(* IEC 61131-3 sources: repolevel_ST_code_completion/output/0127完整版本_带planner/repoeval_VisuElements/readful_result_no_provide, 3 files *)

(* ---- MouseEventHandler.st ---- *)
VAR
    LeftClickTimer : TON;
    xLeftClickOld : BOOL;
    iClickCount : INT := 0;
    xEventProcessed : BOOL := FALSE;
    rLastMouseX : REAL := 0.0;
    rLastMouseY : REAL := 0.0;
END_VAR

(* Reset event state *)
eMouseEvent := 0;
xEventActive := FALSE;

(* Handle left click events (single/double click) *)
IF xLeftClick AND NOT xLeftClickOld THEN
    (* First click detected *)
    IF iClickCount = 0 THEN
        LeftClickTimer(IN := TRUE, PT := tDblClickTime);
        iClickCount := 1;
    ELSE
        (* Second click within time window *)
        LeftClickTimer(IN := FALSE);
        eMouseEvent := 2; (* Double click *)
        rEventX := rMouseX;
        rEventY := rMouseY;
        xEventActive := TRUE;
        iClickCount := 0;
        xEventProcessed := TRUE;
    END_IF
ELSIF NOT xLeftClick AND xLeftClickOld THEN
    (* Left button released *)
    IF iClickCount = 1 AND NOT xEventProcessed THEN
        LeftClickTimer();
        IF NOT LeftClickTimer.Q THEN
            (* Still waiting for potential double click *)
        ELSE
            (* Timeout, register single click *)
            eMouseEvent := 1; (* Single click *)
            rEventX := rMouseX;
            rEventY := rMouseY;
            xEventActive := TRUE;
            iClickCount := 0;
        END_IF
    END_IF
END_IF

(* Check for double click timeout *)
IF LeftClickTimer.Q AND iClickCount = 1 THEN
    (* Timeout, register single click *)
    eMouseEvent := 1; (* Single click *)
    rEventX := rMouseX;
    rEventY := rMouseY;
    xEventActive := TRUE;
    iClickCount := 0;
END_IF

(* Handle right click events *)
IF xRightClick THEN
    eMouseEvent := 3; (* Right click *)
    rEventX := rMouseX;
    rEventY := rMouseY;
    xEventActive := TRUE;
END_IF

(* Handle middle click events *)
IF xMiddleClick THEN
    eMouseEvent := 4; (* Middle click *)
    rEventX := rMouseX;
    rEventY := rMouseY;
    xEventActive := TRUE;
END_IF

(* Handle mouse movement events *)
IF xMouseMove AND (rMouseX <> rLastMouseX OR rMouseY <> rLastMouseY) THEN
    eMouseEvent := 0; (* Mouse move *)
    rEventX := rMouseX;
    rEventY := rMouseY;
    xEventActive := TRUE;
    rLastMouseX := rMouseX;
    rLastMouseY := rMouseY;
END_IF

(* Update old state *)
xLeftClickOld := xLeftClick;
END_FUNCTION_BLOCK

(* ---- NodeExpandCollapse.st ---- *)
VAR
    NodeDblClick : TON; (* Timer for detecting double click *)
    xNodeClickOld : BOOL; (* Previous state of the click input *)
    iNodeState : INT := 1; (* State machine variable *)
END_VAR

CASE iNodeState OF

    1: (* Wait for first click *)
        IF xNodeClick AND NOT xNodeClickOld THEN
            NodeDblClick(IN := TRUE, PT := tDblClickTime);
            iNodeState := 2;
            xNodeSelected := TRUE;
        END_IF

    2: (* Wait for second click or timeout *)
        NodeDblClick();
        IF NodeDblClick.Q THEN
            (* Timeout - single click, reset *)
            NodeDblClick(IN := FALSE);
            xNodeClickOld := FALSE;
            iNodeState := 1;
            xNodeSelected := FALSE;
        ELSIF NOT xNodeClick AND xNodeClickOld THEN
            (* Second click detected - toggle expansion *)
            NodeDblClick(IN := FALSE);
            xNodeExpand := NOT xNodeExpand;
            iNodeState := 1;
            xNodeSelected := FALSE;
        END_IF

END_CASE

xNodeClickOld := xNodeClick;
END_FUNCTION_BLOCK

(* ---- RotationCalculation.st ---- *)
VAR
    rRadians : REAL;
    rCos : REAL;
    rSin : REAL;
    rTranslatedX : REAL;
    rTranslatedY : REAL;
END_VAR

rRadians := rAngle * 3.14159265358979 / 180.0; // Convert angle from degrees to radians
rCos := COS(rRadians);          (* Calculate cosine of the angle *)
rSin := SIN(rRadians);          (* Calculate sine of the angle *)

rTranslatedX := rPointX - rCenterX; (* Calculate relative X coordinate *)
rTranslatedY := rPointY - rCenterY; (* Calculate relative Y coordinate *)

rRotatedX := (rTranslatedX * rCos) - (rTranslatedY * rSin) + rCenterX; (* Calculate rotated X coordinate *)
rRotatedY := (rTranslatedX * rSin) + (rTranslatedY * rCos) + rCenterY; (* Calculate rotated Y coordinate *)

RotationCalculation := TRUE; // Assign return value
RETURN; // End function execution
END_FUNCTION
